FUNCTION F_Variable_TODevice: BOOL

;

END_FUNCTION

(* stored: Version 1.1.0.1, ProductVersion 3.1.4024.15
   POU F_Variable_TODevice: Id {1558be8f-9973-41de-9276-f8ff9a055571}, SpecialFunc None *)
